Universal Robots URScript: proiecFinalHILT_cri.script

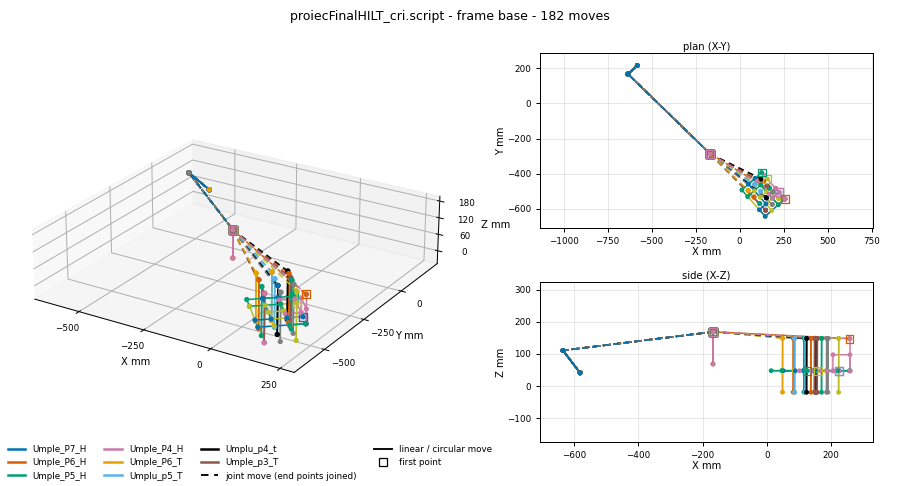
[picture p0: tool path of proiecFinalHILT_cri.script in frame base, 182 of 182 moves have a stored position in this frame; points joined in program order, loops and branches not executed]
def proiecFinalHILT_cri():
  set_gravity([0.0, 0.0, 9.82])
  set_safety_mode_transition_hardness(1)
  set_tool_voltage(24)
  set_tcp(p[0.0,0.0,0.27041000000000004,0.0,0.0,0.0])
  set_payload(0.9, [0.0, 0.0, 0.17])
  set_standard_analog_input_domain(0, 1)
  set_standard_analog_input_domain(1, 1)
  set_tool_analog_input_domain(0, 1)
  set_tool_analog_input_domain(1, 1)
  set_analog_outputdomain(0, 0)
  set_analog_outputdomain(1, 0)
  set_input_actions_to_default()
  step_count_8b5a3645_88be_4d1b_a3a9_0bb7bcbc2ce0 = 0.0
  thread Step_Counter_Thread_93ffaa2a_25e0_4f6a_ae18_d9d09f0d3b97():
    while (True):
      step_count_8b5a3645_88be_4d1b_a3a9_0bb7bcbc2ce0 = step_count_8b5a3645_88be_4d1b_a3a9_0bb7bcbc2ce0 + 1.0
      sync()
    end
  end
  run Step_Counter_Thread_93ffaa2a_25e0_4f6a_ae18_d9d09f0d3b97()
  global poz_switch=3
  global Dist_cub=80
  global countt=2
  global lp=5
  global i_var_1=6
  global Cub=p[-0.5333733899169065,0.2215163955594962,0.16621704113782268,0.29676891717628096,-0.762003058255801,0.6932450754498153]
  global Masa=p[-0.5646864889252723,-0.09295846005778519,-0.011586725889142446,-0.002204506099067434,-1.5199745422116683E-4,-0.8484235711542728]
  global Perete=p[0.07880424455785079,-0.9029855161661187,0.02758526437122058,1.5020481596863833,0.5702478707698211,0.5632393139112222]
  global plan_masa=p[-0.5631648595800378,-0.0915378818255476,-0.042707498643383746,-0.004205331887450723,8.438780583721072E-4,-0.8451230678381721]
  def Umple_P7_H():
    $ 52 "Umple_P7_H" "noBreak"
    $ 53 "MoveJ"
    $ 54 "INTERMED_P7_H" "breakAfter"
    movej(get_inverse_kin(p[-.167567487318, -.286498978533, .168810821008, 1.290941150555, 2.847903107563, -.014389347024], qnear=[0.6869624853134155, -1.9919636885272425, 1.8788256645202637, -1.4593976179706019, -1.5535171667682093, -0.03263694444765264]), a=1.3962634015954636, v=1.0471975511965976)
    $ 55 "Wait: 0.5"
    sleep(0.5)
    $ 56 "MoveJ"
    $ 57 "DEAS_C7_H" "breakAfter"
    movej(get_inverse_kin(p[-.634048678821, .166752753814, .111017315668, 1.076095386128, 2.388610774545, 1.006493672938], qnear=[-0.13465482393373662, -0.5505560080157679, 0.2975288927555084, -0.7133148352252405, -2.1372297445880335, -0.6779091993915003]), a=1.3962634015954636, v=1.0471975511965976)
    $ 58 "Wait: 0.5"
    sleep(0.5)
    $ 59 "MoveL"
    $ 60 "PREL_C7_H" "breakAfter"
    movel(p[-.580966948563, .215040941302, .041371233320, 1.076095361124, 2.388610928008, 1.006493864198], a=1.2, v=0.25)
    $ 61 "Wait: 0.5"
    sleep(0.5)
    $ 62 "'G40'"
    # 'G40'
    $ 63 "MoveL"
    $ 64 "DEAS_C7_HH" "breakAfter"
    movel(p[-.634048678821, .166752753814, .111017315668, 1.076095386128, 2.388610774545, 1.006493672938], a=1.2, v=0.25)
    $ 65 "Wait: 0.5"
    sleep(0.5)
    $ 66 "MoveJ"
    $ 67 "intermed" "breakAfter"
    movej(get_inverse_kin(p[-.167567487318, -.286498978533, .168810821008, 1.290941150555, 2.847903107563, -.014389347024], qnear=[0.6869624853134155, -1.9919636885272425, 1.8788256645202637, -1.4593976179706019, -1.5535171667682093, -0.03263694444765264]), a=1.3962634015954636, v=1.0471975511965976)
    $ 68 "Wait: 0.5"
    sleep(0.5)
    $ 69 "MoveJ"
    $ 70 "DEAS_P7_H_FOAIE" "breakAfter"
    movej(get_inverse_kin(p[.152399925349, -.536216503558, .148554934455, 1.291226875826, 2.847366244409, -.014273160143], qnear=[1.6449040174484253, -1.443597141896383, 1.4715391397476196, -1.6139887014972132, -1.5619214216815394, 0.9256654977798462]), a=1.3962634015954636, v=1.0471975511965976)
    $ 71 "Wait: 0.5"
    sleep(0.5)
    $ 72 "MoveJ"
    $ 73 "LAS_P7_H_FOAIE" "breakAfter"
    movej(get_inverse_kin(p[.151994766277, -.536783252620, -.018790607241, 1.291226898298, 2.847366305883, -.014273512506], qnear=[1.6440799236297607, -1.3487656752215784, 1.8007179498672485, -2.0379918257342737, -1.561909023915426, 0.9248414635658264]), a=1.3962634015954636, v=1.0471975511965976)
    $ 74 "Wait: 0.5"
    sleep(0.5)
    $ 75 "'G 80'"
    # 'G 80'
    $ 76 "MoveL"
    $ 77 "DEAS_C7_H_FOAIE" "breakAfter"
    movel(p[.152399925349, -.536216503558, .148554934455, 1.291226875826, 2.847366244409, -.014273160143], a=1.2, v=0.25)
  end
  def Umple_P6_H():
    $ 78 "Umple_P6_H" "noBreak"
    $ 79 "MoveJ"
    $ 80 "INTERM_C6_H" "breakAfter"
    movej(get_inverse_kin(p[-.167567487318, -.286498978533, .168810821008, 1.290941150555, 2.847903107563, -.014389347024], qnear=[0.6869624853134155, -1.9919636885272425, 1.8788256645202637, -1.4593976179706019, -1.5535171667682093, -0.03263694444765264]), a=1.3962634015954636, v=1.0471975511965976)
    $ 81 "Wait: 0.5"
    sleep(0.5)
    $ 82 "MoveJ"
    $ 83 "DEAS_C6_H" "breakAfter"
    movej(get_inverse_kin(p[-.634048678821, .166752753814, .111017315668, 1.076095386128, 2.388610774545, 1.006493672938], qnear=[-0.13465482393373662, -0.5505560080157679, 0.2975288927555084, -0.7133148352252405, -2.1372297445880335, -0.6779091993915003]), a=1.3962634015954636, v=1.0471975511965976)
    $ 84 "Wait: 0.5"
    sleep(0.5)
    $ 85 "MoveL"
    $ 86 "PREL_C6_H" "breakAfter"
    movel(p[-.580966948563, .215040941302, .041371233320, 1.076095361124, 2.388610928008, 1.006493864198], a=1.2, v=0.25)
    $ 87 "Wait: 0.5"
    sleep(0.5)
    $ 88 "'G40'"
    # 'G40'
    $ 89 "MoveL"
    $ 90 "DEAS_C6_HH" "breakAfter"
    movel(p[-.634048678821, .166752753814, .111017315668, 1.076095386128, 2.388610774545, 1.006493672938], a=1.2, v=0.25)
    $ 91 "Wait: 0.5"
    sleep(0.5)
    $ 92 "MoveJ"
    $ 93 "INTERMEDIARR" "breakAfter"
    movej(get_inverse_kin(p[-.167567487318, -.286498978533, .168810821008, 1.290941150555, 2.847903107563, -.014389347024], qnear=[0.6869624853134155, -1.9919636885272425, 1.8788256645202637, -1.4593976179706019, -1.5535171667682093, -0.03263694444765264]), a=1.3962634015954636, v=1.0471975511965976)
    $ 94 "Wait: 0.5"
    sleep(0.5)
    $ 95 "MoveJ"
    $ 96 "DEAS_P6_H_FOAIE" "breakAfter"
    movej(get_inverse_kin(p[.081815537007, -.531995464645, .148711679169, 2.983820748964, .973323486254, -.005655071201], qnear=[1.5207152366638184, -1.4787958304034632, 1.5076936483383179, -1.6038115660296839, -1.5730794111834925, 2.4608724117279053]), a=1.3962634015954636, v=1.0471975511965976)
    $ 97 "Wait: 0.5"
    sleep(0.5)
    $ 98 "MoveL"
    $ 99 "LAS_P6_H_FOAIE" "breakAfter"
    movel(p[.081410644423, -.532561926736, -.018634025734, 2.983821082689, .973324781842, -.005655577080], a=1.2, v=0.25)
    $ 100 "Wait: 0.5"
    sleep(0.5)
    $ 101 "'G 80'"
    # 'G 80'
    $ 102 "MoveL"
    $ 103 "DEAS_C6_H_FOAIE" "breakAfter"
    movel(p[.081815486859, -.531995349178, .148711350252, 2.983819433937, .973322093540, -.005646498257], a=1.2, v=0.25)
    $ 104 "Wait: 0.5"
    sleep(0.5)
  end
  def Umple_P5_H():
    $ 105 "Umple_P5_H" "noBreak"
    $ 106 "MoveJ"
    $ 107 "INTERM_P5_H" "breakAfter"
    movej(get_inverse_kin(p[-.167567487318, -.286498978533, .168810821008, 1.290941150555, 2.847903107563, -.014389347024], qnear=[0.6869624853134155, -1.9919636885272425, 1.8788256645202637, -1.4593976179706019, -1.5535171667682093, -0.03263694444765264]), a=1.3962634015954636, v=1.0471975511965976)
    $ 108 "Wait: 0.5"
    sleep(0.5)
    $ 109 "MoveJ"
    $ 110 "DEAS_C5_H" "breakAfter"
    movej(get_inverse_kin(p[-.634048678821, .166752753814, .111017315668, 1.076095386128, 2.388610774545, 1.006493672938], qnear=[-0.13465482393373662, -0.5505560080157679, 0.2975288927555084, -0.7133148352252405, -2.1372297445880335, -0.6779091993915003]), a=1.3962634015954636, v=1.0471975511965976)
    $ 111 "Wait: 0.5"
    sleep(0.5)
    $ 112 "MoveL"
    $ 113 "PREL_C5_H" "breakAfter"
    movel(p[-.580966948563, .215040941302, .041371233320, 1.076095361124, 2.388610928008, 1.006493864198], a=1.2, v=0.25)
    $ 114 "Wait: 0.5"
    sleep(0.5)
    $ 115 "'G40'"
    # 'G40'
    $ 116 "MoveL"
    $ 117 "DEAS_C5_HH" "breakAfter"
    movel(p[-.634048678821, .166752753814, .111017315668, 1.076095386128, 2.388610774545, 1.006493672938], a=1.2, v=0.25)
    $ 118 "Wait: 0.5"
    sleep(0.5)
    $ 119 "MoveJ"
    $ 120 "inter" "breakAfter"
    movej(get_inverse_kin(p[-.167567487318, -.286498978533, .168810821008, 1.290941150555, 2.847903107563, -.014389347024], qnear=[0.6869624853134155, -1.9919636885272425, 1.8788256645202637, -1.4593976179706019, -1.5535171667682093, -0.03263694444765264]), a=1.3962634015954636, v=1.0471975511965976)
    $ 121 "Wait: 0.5"
    sleep(0.5)
    $ 122 "MoveJ"
    $ 123 "DEAS_P5_H_FOAIE" "breakAfter"
    movej(get_inverse_kin(p[.114997524645, -.569397994153, .148757924677, 2.983821051292, .973323637050, -.005654878888], qnear=[1.582621455192566, -1.3755558172809046, 1.388292908668518, -1.587501351033346, -1.5733297506915491, 2.522778272628784]), a=1.3962634015954636, v=1.0471975511965976)
    $ 124 "Wait: 0.5"
    sleep(0.5)
    $ 125 "MoveL"
    $ 126 "LAS_P5_H_FOAIE" "breakAfter"
    movel(p[.114592639963, -.569964547732, -.018587646533, 2.983820983248, .973324799820, -.005655526622], a=1.2, v=0.25)
    $ 127 "Wait: 0.5"
    sleep(0.5)
    $ 128 "'G 80'"
    # 'G 80'
    $ 129 "MoveL"
    $ 130 "DEAS_C5_H_FOAIE" "breakAfter"
    movel(p[.114997433899, -.569398004731, .148757767474, 2.983819195458, .973322065302, -.005646601422], a=1.2, v=0.25)
    $ 131 "Wait: 0.5"
    sleep(0.5)
  end
  def Umple_P4_H():
    $ 132 "Umple_P4_H" "noBreak"
    $ 133 "MoveJ"
    $ 134 "INTERM_P4_H" "breakAfter"
    movej(get_inverse_kin(p[-.167567487318, -.286498978533, .168810821008, 1.290941150555, 2.847903107563, -.014389347024], qnear=[0.6869624853134155, -1.9919636885272425, 1.8788256645202637, -1.4593976179706019, -1.5535171667682093, -0.03263694444765264]), a=1.3962634015954636, v=1.0471975511965976)
    $ 135 "Wait: 0.5"
    sleep(0.5)
    $ 136 "MoveJ"
    $ 137 "DEAS_C4_H" "breakAfter"
    movej(get_inverse_kin(p[-.634048678821, .166752753814, .111017315668, 1.076095386128, 2.388610774545, 1.006493672938], qnear=[-0.13465482393373662, -0.5505560080157679, 0.2975288927555084, -0.7133148352252405, -2.1372297445880335, -0.6779091993915003]), a=1.3962634015954636, v=1.0471975511965976)
    $ 138 "Wait: 0.5"
    sleep(0.5)
    $ 139 "MoveL"
    $ 140 "PREL_C4_H" "breakAfter"
    movel(p[-.580966948563, .215040941302, .041371233320, 1.076095361124, 2.388610928008, 1.006493864198], a=1.2, v=0.25)
    $ 141 "Wait: 0.5"
    sleep(0.5)
    $ 142 "'G40'"
    # 'G40'
    $ 143 "MoveL"
    $ 144 "DEAS_C4_HH" "breakAfter"
    movel(p[-.634048678821, .166752753814, .111017315668, 1.076095386128, 2.388610774545, 1.006493672938], a=1.2, v=0.25)
    $ 145 "Wait: 0.5"
    sleep(0.5)
    $ 146 "MoveJ"
    $ 147 "INTERMEDIA" "breakAfter"
    movej(get_inverse_kin(p[-.167567487318, -.286498978533, .168810821008, 1.290941150555, 2.847903107563, -.014389347024], qnear=[0.6869624853134155, -1.9919636885272425, 1.8788256645202637, -1.4593976179706019, -1.5535171667682093, -0.03263694444765264]), a=1.3962634015954636, v=1.0471975511965976)
    $ 148 "Wait: 0.5"
    sleep(0.5)
    $ 149 "MoveJ"
    $ 150 "DEAS_P4_H_FOAIE" "breakAfter"
    movej(get_inverse_kin(p[.148179526257, -.606800607225, .148804148337, 2.983821216675, .973323524331, -.005654610012], qnear=[1.6362345218658447, -1.2673490683185022, 1.2510157823562622, -1.5582893530475062, -1.573538605366842, 2.5763912200927734]), a=1.3962634015954636, v=1.0471975511965976)
    $ 151 "Wait: 0.5"
    sleep(0.5)
    $ 152 "MoveL"
    $ 153 "LAS_P4_H_FOAIE" "breakAfter"
    movel(p[.147774535974, -.607367175758, -.018541400911, 2.983821119944, .973324675130, -.005655864895], a=1.2, v=0.25)
    $ 154 "Wait: 0.5"
    sleep(0.5)
    $ 155 "'G 80'"
    # 'G 80'
    $ 156 "MoveL"
    $ 157 "DEAS_P4_H" "breakAfter"
    movel(p[.148179486526, -.606800539344, .148804102555, 2.983819245133, .973322110034, -.005646290070], a=1.2, v=0.25)
    $ 158 "Wait: 0.5"
    sleep(0.5)
  end
  def Umple_P6_T():
    $ 159 "Umple_P6_T" "noBreak"
    $ 160 "MoveJ"
    $ 161 "INTERM_C6_T" "breakAfter"
    movej(get_inverse_kin(p[-.167567487318, -.286498978533, .168810821008, 1.290941150555, 2.847903107563, -.014389347024], qnear=[0.6869624853134155, -1.9919636885272425, 1.8788256645202637, -1.4593976179706019, -1.5535171667682093, -0.03263694444765264]), a=1.3962634015954636, v=1.0471975511965976)
    $ 162 "Wait: 0.5"
    sleep(0.5)
    $ 163 "MoveJ"
    $ 164 "DEAS_C6_T" "breakAfter"
    movej(get_inverse_kin(p[-.634048678821, .166752753814, .111017315668, 1.076095386128, 2.388610774545, 1.006493672938], qnear=[-0.13465482393373662, -0.5505560080157679, 0.2975288927555084, -0.7133148352252405, -2.1372297445880335, -0.6779091993915003]), a=1.3962634015954636, v=1.0471975511965976)
    $ 165 "Wait: 0.5"
    sleep(0.5)
    $ 166 "MoveL"
    $ 167 "PREL_C6_T" "breakAfter"
    movel(p[-.580966948563, .215040941302, .041371233320, 1.076095361124, 2.388610928008, 1.006493864198], a=1.2, v=0.25)
    $ 168 "Wait: 0.5"
    sleep(0.5)
    $ 169 "'G40'"
    # 'G40'
    $ 170 "MoveL"
    $ 171 "DEAS_C6_TT" "breakAfter"
    movel(p[-.634048678821, .166752753814, .111017315668, 1.076095386128, 2.388610774545, 1.006493672938], a=1.2, v=0.25)
    $ 172 "Wait: 0.5"
    sleep(0.5)
    $ 173 "MoveJ"
    $ 174 "INTERME" "breakAfter"
    movej(get_inverse_kin(p[-.167567487318, -.286498978533, .168810821008, 1.290941150555, 2.847903107563, -.014389347024], qnear=[0.6869624853134155, -1.9919636885272425, 1.8788256645202637, -1.4593976179706019, -1.5535171667682093, -0.03263694444765264]), a=1.3962634015954636, v=1.0471975511965976)
    $ 175 "Wait: 0.5"
    sleep(0.5)
    $ 176 "MoveJ"
    $ 177 "DEAS_P6_T_FOAIE" "breakAfter"
    movej(get_inverse_kin(p[.086036154554, -.461411134347, .148462036457, 2.983821038078, .973324356096, -.005654006834], qnear=[1.5222129821777344, -1.644914452229635, 1.676056146621704, -1.606051270161764, -1.573085133229391, 2.462369680404663]), a=1.3962634015954636, v=1.0471975511965976)
    $ 178 "Wait: 0.5"
    sleep(0.5)
    $ 179 "MoveL"
    $ 180 "LAS_C6_T_FOAIE" "breakAfter"
    movel(p[.085630996758, -.461978027654, -.018883318685, 2.983820678969, .973324049014, -.005654378319], a=1.2, v=0.25)
    $ 181 "Wait: 0.5"
    sleep(0.5)
    $ 182 "'G 80'"
    # 'G 80'
    $ 183 "MoveL"
    $ 184 "DEAS_P6_T" "breakAfter"
    movel(p[.086036154554, -.461411134347, .148462036457, 2.983821038078, .973324356096, -.005654006834], a=1.2, v=0.25)
    $ 185 "Wait: 0.5"
    sleep(0.5)
  end
  def Umplu_p5_T():
    $ 186 "Umplu_p5_T" "noBreak"
    $ 187 "MoveJ"
    $ 188 "INTERM_P5_T" "breakAfter"
    movej(get_inverse_kin(p[-.167567487318, -.286498978533, .168810821008, 1.290941150555, 2.847903107563, -.014389347024], qnear=[0.6869624853134155, -1.9919636885272425, 1.8788256645202637, -1.4593976179706019, -1.5535171667682093, -0.03263694444765264]), a=1.3962634015954636, v=1.0471975511965976)
    $ 189 "Wait: 0.5"
    sleep(0.5)
    $ 190 "MoveJ"
    $ 191 "DEAS_C5_T" "breakAfter"
    movej(get_inverse_kin(p[-.634048678821, .166752753814, .111017315668, 1.076095386128, 2.388610774545, 1.006493672938], qnear=[-0.13465482393373662, -0.5505560080157679, 0.2975288927555084, -0.7133148352252405, -2.1372297445880335, -0.6779091993915003]), a=1.3962634015954636, v=1.0471975511965976)
    $ 192 "Wait: 0.5"
    sleep(0.5)
    $ 193 "MoveL"
    $ 194 "PREL_C5_T" "breakAfter"
    movel(p[-.580966948563, .215040941302, .041371233320, 1.076095361124, 2.388610928008, 1.006493864198], a=1.2, v=0.25)
    $ 195 "Wait: 0.5"
    sleep(0.5)
    $ 196 "'G40'"
    # 'G40'
    $ 197 "MoveL"
    $ 198 "DEAS_C5_TT" "breakAfter"
    movel(p[-.634048678821, .166752753814, .111017315668, 1.076095386128, 2.388610774545, 1.006493672938], a=1.2, v=0.25)
    $ 199 "Wait: 0.5"
    sleep(0.5)
    $ 200 "MoveJ"
    $ 201 "INter" "breakAfter"
    movej(get_inverse_kin(p[-.167567487318, -.286498978533, .168810821008, 1.290941150555, 2.847903107563, -.014389347024], qnear=[0.6869624853134155, -1.9919636885272425, 1.8788256645202637, -1.4593976179706019, -1.5535171667682093, -0.03263694444765264]), a=1.3962634015954636, v=1.0471975511965976)
    $ 202 "Wait: 0.5"
    sleep(0.5)
    $ 203 "MoveJ"
    $ 204 "DEAS_P5_T_FOAIE" "breakAfter"
    movej(get_inverse_kin(p[.119218109273, -.498813767404, .148508400157, 2.983820953563, .973324318096, -.005654075141], qnear=[1.592743992805481, -1.5396392981158655, 1.5730714797973633, -1.6081703344928187, -1.57336932817568, 2.532900333404541]), a=1.3962634015954636, v=1.0471975511965976)
    $ 205 "Wait: 0.5"
    sleep(0.5)
    $ 206 "MoveL"
    $ 207 "LAS_C5_T_FOAIE" "breakAfter"
    movel(p[.118812995133, -.499380619453, -.018837005131, 2.983820836474, .973323892156, -.005654109965], a=1.2, v=0.25)
    $ 208 "Wait: 0.5"
    sleep(0.5)
    $ 209 "'G 80'"
    # 'G 80'
    $ 210 "MoveL"
    $ 211 "DEAS_P5" "breakAfter"
    movel(p[.119218109273, -.498813767404, .148508400157, 2.983820953563, .973324318096, -.005654075141], a=1.2, v=0.25)
    $ 212 "Wait: 0.5"
    sleep(0.5)
  end
  def Umplu_p4_t():
    $ 213 "Umplu_p4_t" "noBreak"
    $ 214 "MoveJ"
    $ 215 "interm_p4_t" "breakAfter"
    movej(get_inverse_kin(p[-.167567487318, -.286498978533, .168810821008, 1.290941150555, 2.847903107563, -.014389347024], qnear=[0.6869624853134155, -1.9919636885272425, 1.8788256645202637, -1.4593976179706019, -1.5535171667682093, -0.03263694444765264]), a=1.3962634015954636, v=1.0471975511965976)
    $ 216 "Wait: 0.5"
    sleep(0.5)
    $ 217 "MoveJ"
    $ 218 "deas_c4_T" "breakAfter"
    movej(get_inverse_kin(p[-.634048678821, .166752753814, .111017315668, 1.076095386128, 2.388610774545, 1.006493672938], qnear=[-0.13465482393373662, -0.5505560080157679, 0.2975288927555084, -0.7133148352252405, -2.1372297445880335, -0.6779091993915003]), a=1.3962634015954636, v=1.0471975511965976)
    $ 219 "Wait: 0.5"
    sleep(0.5)
    $ 220 "MoveL"
    $ 221 "PREL_C4_T" "breakAfter"
    movel(p[-.580966948563, .215040941302, .041371233320, 1.076095361124, 2.388610928008, 1.006493864198], a=1.2, v=0.25)
    $ 222 "Wait: 0.5"
    sleep(0.5)
    $ 223 "'G40'"
    # 'G40'
    $ 224 "MoveL"
    $ 225 "DEAS_C4_T" "breakAfter"
    movel(p[-.634048678821, .166752753814, .111017315668, 1.076095386128, 2.388610774545, 1.006493672938], a=1.2, v=0.25)
    $ 226 "Wait: 0.5"
    sleep(0.5)
    $ 227 "MoveJ"
    $ 228 "INTERMEDIAR" "breakAfter"
    movej(get_inverse_kin(p[-.167567487318, -.286498978533, .168810821008, 1.290941150555, 2.847903107563, -.014389347024], qnear=[0.6869624853134155, -1.9919636885272425, 1.8788256645202637, -1.4593976179706019, -1.5535171667682093, -0.03263694444765264]), a=1.3962634015954636, v=1.0471975511965976)
    $ 229 "Wait: 0.5"
    sleep(0.5)
    $ 230 "MoveJ"
    $ 231 "DEAS_P4_T_FOAIE" "breakAfter"
    movej(get_inverse_kin(p[.152399990844, -.536216423213, .148554701618, 2.983821087416, .973324179283, -.005654354735], qnear=[1.652442216873169, -1.4321559111224573, 1.4555567502975464, -1.597978417073385, -1.5736001173602503, 2.5925984382629395]), a=1.3962634015954636, v=1.0471975511965976)
    $ 232 "Wait: 0.5"
    sleep(0.5)
    $ 233 "MoveL"
    $ 234 "LAS_P4_T_FOAIE" "breakAfter"
    movel(p[.151994974835, -.536783166276, -.018790624961, 2.983820916063, .973323931244, -.005654087772], a=1.2, v=0.25)
    $ 235 "Wait: 0.5"
    sleep(0.5)
    $ 236 "'G 80'"
    # 'G 80'
    $ 237 "MoveL"
    $ 238 "DEAS_P4_T" "breakAfter"
    movel(p[.152399990844, -.536216423213, .148554701618, 2.983821087416, .973324179283, -.005654354735], a=1.2, v=0.25)
    $ 239 "Wait: 0.5"
    sleep(0.5)
  end
  def Umple_p3_T():
    $ 240 "Umple_p3_T" "noBreak"
    $ 241 "MoveJ"
    $ 242 "INTERM_P3_T" "breakAfter"
    movej(get_inverse_kin(p[-.167567487318, -.286498978533, .168810821008, 1.290941150555, 2.847903107563, -.014389347024], qnear=[0.6869624853134155, -1.9919636885272425, 1.8788256645202637, -1.4593976179706019, -1.5535171667682093, -0.03263694444765264]), a=1.3962634015954636, v=1.0471975511965976)
    $ 243 "Wait: 0.5"
    sleep(0.5)
    $ 244 "MoveJ"
    $ 245 "DEAS_C3_T" "breakAfter"
    movej(get_inverse_kin(p[-.634048678821, .166752753814, .111017315668, 1.076095386128, 2.388610774545, 1.006493672938], qnear=[-0.13465482393373662, -0.5505560080157679, 0.2975288927555084, -0.7133148352252405, -2.1372297445880335, -0.6779091993915003]), a=1.3962634015954636, v=1.0471975511965976)
    $ 246 "Wait: 0.5"
    sleep(0.5)
    $ 247 "MoveL"
    $ 248 "PREL_C3_T" "breakAfter"
    movel(p[-.580966948563, .215040941302, .041371233320, 1.076095361124, 2.388610928008, 1.006493864198], a=1.2, v=0.25)
    $ 249 "Wait: 0.5"
    sleep(0.5)
    $ 250 "'G40'"
    # 'G40'
    $ 251 "MoveL"
    $ 252 "DEAS_C3_TT" "breakAfter"
    movel(p[-.634048678821, .166752753814, .111017315668, 1.076095386128, 2.388610774545, 1.006493672938], a=1.2, v=0.25)
    $ 253 "Wait: 0.5"
    sleep(0.5)
    $ 254 "MoveJ"
    $ 255 "INTERMEDD" "breakAfter"
    movej(get_inverse_kin(p[-.167567487318, -.286498978533, .168810821008, 1.290941150555, 2.847903107563, -.014389347024], qnear=[0.6869624853134155, -1.9919636885272425, 1.8788256645202637, -1.4593976179706019, -1.5535171667682093, -0.03263694444765264]), a=1.3962634015954636, v=1.0471975511965976)
    $ 256 "Wait: 0.5"
    sleep(0.5)
    $ 257 "MoveJ"
    $ 258 "DEAS_P3_T_FOAIE" "breakAfter"
    movej(get_inverse_kin(p[.148179528223, -.606800592740, .148804018507, 1.291225298432, 2.847366483862, -.014273607498], qnear=[1.6294351816177368, -1.2790477911578577, 1.2692852020263672, -1.5761454741107386, -1.5616863409625452, 0.910196840763092]), a=1.3962634015954636, v=1.0471975511965976)
    $ 259 "Wait: 0.5"
    sleep(0.5)
    $ 260 "MoveL"
    $ 261 "LAS_P3_T_FOAIE" "breakAfter"
    movel(p[.147774525895, -.607367213899, -.018541509057, 1.291225168160, 2.847366616510, -.014273004499], a=1.2, v=0.25)
    $ 262 "Wait: 0.5"
    sleep(0.5)
    $ 263 "'G 80'"
    # 'G 80'
    $ 264 "MoveL"
    $ 265 "DEAS_P3_T" "breakAfter"
    movel(p[.148179528223, -.606800592740, .148804018507, 1.291225298432, 2.847366483862, -.014273607498], a=1.2, v=0.25)
    $ 266 "Wait: 0.5"
    sleep(0.5)
  end
  def Umple_P2_T():
    $ 267 "Umple_P2_T" "noBreak"
    $ 268 "MoveJ"
    $ 269 "INTERM_P2_T" "breakAfter"
    movej(get_inverse_kin(p[-.167567487318, -.286498978533, .168810821008, 1.290941150555, 2.847903107563, -.014389347024], qnear=[0.6869624853134155, -1.9919636885272425, 1.8788256645202637, -1.4593976179706019, -1.5535171667682093, -0.03263694444765264]), a=1.3962634015954636, v=1.0471975511965976)
    $ 270 "Wait: 0.5"
    sleep(0.5)
    $ 271 "MoveJ"
    $ 272 "DEAS_P2_T" "breakAfter"
    movej(get_inverse_kin(p[-.634048678821, .166752753814, .111017315668, 1.076095386128, 2.388610774545, 1.006493672938], qnear=[-0.13465482393373662, -0.5505560080157679, 0.2975288927555084, -0.7133148352252405, -2.1372297445880335, -0.6779091993915003]), a=1.3962634015954636, v=1.0471975511965976)
    $ 273 "Wait: 0.5"
    sleep(0.5)
    $ 274 "MoveL"
    $ 275 "PREL_C2_T" "breakAfter"
    movel(p[-.580966948563, .215040941302, .041371233320, 1.076095361124, 2.388610928008, 1.006493864198], a=1.2, v=0.25)
    $ 276 "Wait: 0.5"
    sleep(0.5)
    $ 277 "'G40'"
    # 'G40'
    $ 278 "MoveL"
    $ 279 "DEAS_C2_T" "breakAfter"
    movel(p[-.634048678821, .166752753814, .111017315668, 1.076095386128, 2.388610774545, 1.006493672938], a=1.2, v=0.25)
    $ 280 "Wait: 0.5"
    sleep(0.5)
    $ 281 "MoveJ"
    $ 282 "INTERMED" "breakAfter"
    movej(get_inverse_kin(p[-.167567487318, -.286498978533, .168810821008, 1.290941150555, 2.847903107563, -.014389347024], qnear=[0.6869624853134155, -1.9919636885272425, 1.8788256645202637, -1.4593976179706019, -1.5535171667682093, -0.03263694444765264]), a=1.3962634015954636, v=1.0471975511965976)
    $ 283 "Wait: 0.5"
    sleep(0.5)
    $ 284 "MoveJ"
    $ 285 "DEAS_P2_T_FOAIE" "breakAfter"
    movej(get_inverse_kin(p[.185581949577, -.573618939446, .148601050831, 1.291225391927, 2.847366587857, -.014273246615], qnear=[1.696845293045044, -1.3333137671100062, 1.339584231376648, -1.592757527028219, -1.5627248922931116, 0.9776014685630798]), a=1.3962634015954636, v=1.0471975511965976)
    $ 286 "Wait: 0.5"
    sleep(0.5)
    $ 287 "MoveL"
    $ 288 "LAS_P2_T_FOAIE" "breakAfter"
    movel(p[.185176974658, -.574185681297, -.018744368520, 1.291225186600, 2.847366418911, -.014273142291], a=1.2, v=0.25)
    $ 289 "Wait: 0.5"
    sleep(0.5)
    $ 290 "'G 80'"
    # 'G 80'
    $ 291 "MoveL"
    $ 292 "DEAS_P2_T_F" "breakAfter"
    movel(p[.185581949577, -.573618939446, .148601050831, 1.291225391927, 2.847366587857, -.014273246615], a=1.2, v=0.25)
    $ 293 "Wait: 0.5"
    sleep(0.5)
  end
  def Desen_H():
    $ 294 "Desen_H" "noBreak"
    $ 295 "MoveL"
    $ 296 "L1_H" "breakAfter"
    movel(p[.158353767573, -.430155299332, .047611332993, 1.296043145667, 2.848527183735, .014471728358], a=1.2, v=0.25)
    $ 297 "MoveL"
    $ 298 "L2_H" "breakAfter"
    movel(p[.120951283833, -.463336924786, .047814223162, 1.296043120148, 2.848527345096, .014471416584], a=1.2, v=0.25)
    $ 299 "MoveL"
    $ 300 "L3_H" "breakAfter"
    movel(p[.154133236674, -.500739444601, .047860495744, 1.296043187324, 2.848527522418, .014471774946], a=1.2, v=0.25)
    $ 301 "MoveL"
    $ 302 "L4_H" "breakAfter"
    movel(p[.116730864622, -.533921061136, .048063444108, 1.296043121592, 2.848527328027, .014471677397], a=1.2, v=0.25)
    $ 303 "MoveL"
    $ 304 "L5_H" "breakAfter"
    movel(p[.083548907102, -.496518450929, .048017030358, 1.296043098946, 2.848527421426, .014471904572], a=1.2, v=0.25)
    $ 305 "MoveL"
    $ 306 "L6_H" "breakAfter"
    movel(p[.046146485395, -.529699970965, .048219970789, 1.296043094495, 2.848527467819, .014471901899], a=1.2, v=0.25)
    $ 307 "MoveL"
    $ 308 "L7_H" "breakAfter"
    movel(p[.145692315173, -.641907763135, .048359070968, 1.296043194804, 2.848527583583, .014471694291], a=1.2, v=0.25)
    $ 309 "MoveL"
    $ 310 "L8" "breakAfter"
    movel(p[.183094788894, -.608726180961, .048156303017, 1.296043066858, 2.848527509527, .014471421053], a=1.2, v=0.25)
    $ 311 "MoveL"
    $ 312 "L9_H" "breakAfter"
    movel(p[.149912797167, -.571323507272, .048109955944, 1.296043112977, 2.848527628353, .014471593212], a=1.2, v=0.25)
    $ 313 "MoveL"
    $ 314 "L10_H" "breakAfter"
    movel(p[.187315154740, -.538141973257, .047906982215, 1.296043228903, 2.848527813831, .014471559318], a=1.2, v=0.25)
    $ 315 "MoveL"
    $ 316 "L11_H" "breakAfter"
    movel(p[.220497113487, -.575544528094, .047953430580, 1.296043230770, 2.848527753786, .014471533520], a=1.2, v=0.25)
    $ 317 "MoveL"
    $ 318 "L12_H" "breakAfter"
    movel(p[.257899491601, -.542362921046, .047750448037, 1.296043415155, 2.848527963236, .014471718970], a=1.2, v=0.25)
  end
  def Desen_T():
    $ 319 "Desen_T" "noBreak"
    $ 320 "MoveL"
    $ 321 "l1_T" "breakAfter"
    movel(p[.224717745310, -.504960528950, .047704168521, 1.296043065165, 2.848526931384, .014471352058], a=1.2, v=0.25)
    $ 322 "MoveL"
    $ 323 "l2_T" "breakAfter"
    movel(p[.187315272317, -.538142086044, .047906973360, 1.296043149277, 2.848527197326, .014471477363], a=1.2, v=0.25)
    $ 324 "MoveL"
    $ 325 "l3_T" "breakAfter"
    movel(p[.087769321683, -.425934317539, .047767997329, 1.296043100195, 2.848527282499, .014471150240], a=1.2, v=0.25)
    $ 326 "MoveL"
    $ 327 "l4_T" "breakAfter"
    movel(p[.050366823128, -.459115956447, .047970927808, 1.296043197593, 2.848527294810, .014470760370], a=1.2, v=0.25)
    $ 328 "MoveL"
    $ 329 "l5_T" "breakAfter"
    movel(p[.149912749792, -.571323861062, .048110045365, 1.296043089492, 2.848527153310, .014470272402], a=1.2, v=0.25)
    $ 330 "MoveL"
    $ 331 "l6_T" "breakAfter"
    movel(p[.112510303828, -.604505478994, .048312930113, 1.296043108336, 2.848527098013, .014470239028], a=1.2, v=0.25)
    $ 332 "MoveL"
    $ 333 "l7_T" "breakAfter"
    movel(p[.145692254958, -.641908116683, .048359160323, 1.296043175969, 2.848527118698, .014470364418], a=1.2, v=0.25)
    $ 334 "MoveL"
    $ 335 "l8_T" "breakAfter"
    movel(p[.257899539344, -.542363388286, .047750527044, 1.296043062532, 2.848527225834, .014470116205], a=1.2, v=0.25)
  end
  def Umplu_p3_i():
    $ 336 "Umplu_p3_i" "noBreak"
    $ 337 "MoveJ"
    $ 338 "interm_p3" "breakAfter"
    movej(get_inverse_kin(p[-.167567487318, -.286498978533, .168810821008, 1.290941150555, 2.847903107563, -.014389347024], qnear=[0.6869624853134155, -1.9919636885272425, 1.8788256645202637, -1.4593976179706019, -1.5535171667682093, -0.03263694444765264]), a=1.3962634015954636, v=1.0471975511965976)
    $ 339 "Wait: 0.5"
    sleep(0.5)
    $ 340 "MoveJ"
    $ 341 "deas_c3_i" "breakAfter"
    movej(get_inverse_kin(p[-.634048678821, .166752753814, .111017315668, 1.076095386128, 2.388610774545, 1.006493672938], qnear=[-0.13465482393373662, -0.5505560080157679, 0.2975288927555084, -0.7133148352252405, -2.1372297445880335, -0.6779091993915003]), a=1.3962634015954636, v=1.0471975511965976)
    $ 342 "Wait: 0.5"
    sleep(0.5)
    $ 343 "MoveL"
    $ 344 "prel_3_i" "breakAfter"
    movel(p[-.580966948563, .215040941302, .041371233320, 1.076095361124, 2.388610928008, 1.006493864198], a=1.2, v=0.25)
    $ 345 "Wait: 0.5"
    sleep(0.5)
    $ 346 "'G40'"
    # 'G40'
    $ 347 "MoveL"
    $ 348 "deas_c3_ii" "breakAfter"
    movel(p[-.634048678821, .166752753814, .111017315668, 1.076095386128, 2.388610774545, 1.006493672938], a=1.2, v=0.25)
    $ 349 "Wait: 0.5"
    sleep(0.5)
    $ 350 "MoveJ"
    $ 351 "interm" "breakAfter"
    movej(get_inverse_kin(p[-.167567487318, -.286498978533, .168810821008, 1.290941150555, 2.847903107563, -.014389347024], qnear=[0.6869624853134155, -1.9919636885272425, 1.8788256645202637, -1.4593976179706019, -1.5535171667682093, -0.03263694444765264]), a=1.3962634015954636, v=1.0471975511965976)
    $ 352 "Wait: 0.5"
    sleep(0.5)
    $ 353 "MoveJ"
    $ 354 "deas_p3_i_foaie" "breakAfter"
    movej(get_inverse_kin(p[.136710917520, -.443190700033, .148277597898, 2.983706779009, .973287613512, -.005232679259], qnear=[1.6343494653701782, -1.6582220236407679, 1.688613772392273, -1.6050694624530237, -1.5732410589801233, 2.5745058059692383]), a=1.3962634015954636, v=1.0471975511965976)
    $ 355 "Wait: 0.5"
    sleep(0.5)
    $ 356 "MoveL"
    $ 357 "las_p3_i_foaie" "breakAfter"
    movel(p[.136306192414, -.443757445123, -.019067699712, 2.983706719795, .973287408143, -.005231154998], a=1.2, v=0.25)
    $ 358 "Wait: 0.5"
    sleep(0.5)
    $ 359 "'G 80'"
    # 'G 80'
    $ 360 "MoveL"
    $ 361 "deas_p3_i" "breakAfter"
    movel(p[.136710967595, -.443190640401, .148277539713, 2.983707061866, .973287115721, -.005232631375], a=1.2, v=0.25)
  end
  def Umplu_p2_i():
    $ 362 "Umplu_p2_i" "noBreak"
    $ 363 "MoveJ"
    $ 364 "interm_p2_i" "breakAfter"
    movej(get_inverse_kin(p[-.167567487318, -.286498978533, .168810821008, 1.290941150555, 2.847903107563, -.014389347024], qnear=[0.6869624853134155, -1.9919636885272425, 1.8788256645202637, -1.4593976179706019, -1.5535171667682093, -0.03263694444765264]), a=1.3962634015954636, v=1.0471975511965976)
    $ 365 "Wait: 0.5"
    sleep(0.5)
    $ 366 "MoveJ"
    $ 367 "deas_c2_i" "breakAfter"
    movej(get_inverse_kin(p[-.634048678821, .166752753814, .111017315668, 1.076095386128, 2.388610774545, 1.006493672938], qnear=[-0.13465482393373662, -0.5505560080157679, 0.2975288927555084, -0.7133148352252405, -2.1372297445880335, -0.6779091993915003]), a=1.3962634015954636, v=1.0471975511965976)
    $ 368 "Wait: 0.5"
    sleep(0.5)
    $ 369 "MoveL"
    $ 370 "prel_c2_i" "breakAfter"
    movel(p[-.580966948563, .215040941302, .041371233320, 1.076095361124, 2.388610928008, 1.006493864198], a=1.2, v=0.25)
    $ 371 "Wait: 0.5"
    sleep(0.5)
    $ 372 "'G40'"
    # 'G40'
    $ 373 "MoveL"
    $ 374 "deas_c2_i2" "breakAfter"
    movel(p[-.634048678821, .166752753814, .111017315668, 1.076095386128, 2.388610774545, 1.006493672938], a=1.2, v=0.25)
    $ 375 "Wait: 0.5"
    sleep(0.5)
    $ 376 "MoveJ"
    $ 377 "intermmm" "breakAfter"
    movej(get_inverse_kin(p[-.167567487318, -.286498978533, .168810821008, 1.290941150555, 2.847903107563, -.014389347024], qnear=[0.6869624853134155, -1.9919636885272425, 1.8788256645202637, -1.4593976179706019, -1.5535171667682093, -0.03263694444765264]), a=1.3962634015954636, v=1.0471975511965976)
    $ 378 "Wait: 0.5"
    sleep(0.5)
    $ 379 "MoveJ"
    $ 380 "Deas_P2_I_FOaie" "breakAfter"
    movej(get_inverse_kin(p[.169892934208, -.480593350924, .148323950518, 2.983706611248, .973287743483, -.005232594662], qnear=[1.696690559387207, -1.54694110551943, 1.5810078382492065, -1.6085847059832972, -1.5734780470477503, 2.6368465423583984]), a=1.3962634015954636, v=1.0471975511965976)
    $ 381 "Wait: 0.5"
    sleep(0.5)
    $ 382 "MoveL"
    $ 383 "las_P2_i_foaie" "breakAfter"
    movel(p[.169488097210, -.481159998853, -.019021462959, 2.983706968312, .973287474864, -.005231319054], a=1.2, v=0.25)
    $ 384 "Wait: 0.5"
    sleep(0.5)
    $ 385 "'G 80'"
    # 'G 80'
    $ 386 "MoveL"
    $ 387 "deas_p2_i" "breakAfter"
    movel(p[.169892986025, -.480593287420, .148323892346, 2.983706895626, .973287246212, -.005232558159], a=1.2, v=0.25)
  end
  def Desen_i():
    $ 388 "Desen_i" "noBreak"
    $ 389 "MoveL"
    $ 390 "Caciulita_i1" "breakAfter"
    movel(p[.224717722166, -.504960484151, .047704103504, 1.291226847034, 2.847366347327, -.014272085334], a=1.2, v=0.25)
    $ 391 "MoveL"
    $ 392 "Caciulita_i2" "breakAfter"
    movel(p[.187315226594, -.538142043484, .047906977082, 1.291227032284, 2.847366301756, -.014272118413], a=1.2, v=0.25)
    $ 393 "MoveL"
    $ 394 "caciulita_i3" "breakAfter"
    movel(p[.220497136640, -.575544671583, .047953560433, 1.291225944203, 2.847366585140, -.014274123381], a=1.2, v=0.25)
    $ 395 "MoveL"
    $ 396 "Caciulita_i4" "breakAfter"
    movel(p[.257899562405, -.542362928148, .047750267064, 1.291226593864, 2.847366752439, -.014272422908], a=1.2, v=0.25)
    $ 397 "MoveL"
    $ 398 "spatiere1_i" "breakAfter"
    movel(p[.258020743673, -.542193728640, .097750042331, 1.291224449561, 2.847366863892, -.014275606648], a=1.2, v=0.25)
    $ 399 "MoveL"
    $ 400 "spatiere2_i" "breakAfter"
    movel(p[.204929683954, -.482349502149, .097676031332, 1.291226728538, 2.847366079793, -.014272245406], a=1.2, v=0.25)
    $ 401 "MoveL"
    $ 402 "spatiere3_i" "breakAfter"
    movel(p[.204808597099, -.482518777578, .047676475167, 1.291226441140, 2.847366455616, -.014273107727], a=1.2, v=0.25)
    $ 403 "MoveL"
    $ 404 "coada_i1" "breakAfter"
    movel(p[.138444723852, -.407713504749, .047583847563, 1.291226332997, 2.847366307920, -.014273010711], a=1.2, v=0.25)
    $ 405 "MoveL"
    $ 406 "coada_i2" "breakAfter"
    movel(p[.101042232951, -.440895027094, .047786740412, 1.291226372130, 2.847366540430, -.014272971580], a=1.2, v=0.25)
    $ 407 "MoveL"
    $ 408 "coada_i3" "breakAfter"
    movel(p[.167406116273, -.515700163940, .047879477850, 1.291226451164, 2.847366681792, -.014273039441], a=1.2, v=0.25)
    $ 409 "MoveL"
    $ 410 "coada_i4" "breakAfter"
    movel(p[.204808616914, -.482518553621, .047676614829, 1.291226300396, 2.847366594866, -.014272954152], a=1.2, v=0.25)
  end
  def Umplu_P6_L():
    $ 411 "Umplu_P6_L" "noBreak"
    $ 412 "MoveJ"
    $ 413 "INTERM_P6" "breakAfter"
    movej(get_inverse_kin(p[-.167567487318, -.286498978533, .168810821008, 1.290941150555, 2.847903107563, -.014389347024], qnear=[0.6869624853134155, -1.9919636885272425, 1.8788256645202637, -1.4593976179706019, -1.5535171667682093, -0.03263694444765264]), a=1.3962634015954636, v=1.0471975511965976)
    $ 414 "Wait: 0.5"
    sleep(0.5)
    $ 415 "MoveJ"
    $ 416 "DEAS_C6_L" "breakAfter"
    movej(get_inverse_kin(p[-.634048678821, .166752753814, .111017315668, 1.076095386128, 2.388610774545, 1.006493672938], qnear=[-0.13465482393373662, -0.5505560080157679, 0.2975288927555084, -0.7133148352252405, -2.1372297445880335, -0.6779091993915003]), a=1.3962634015954636, v=1.0471975511965976)
    $ 417 "Wait: 0.5"
    sleep(0.5)
    $ 418 "MoveL"
    $ 419 "PREL_C6_L" "breakAfter"
    movel(p[-.580966948563, .215040941302, .041371233320, 1.076095361124, 2.388610928008, 1.006493864198], a=1.2, v=0.25)
    $ 420 "Wait: 0.5"
    sleep(0.5)
    $ 421 "'G40'"
    # 'G40'
    $ 422 "MoveL"
    $ 423 "DEAS_C6_LL" "breakAfter"
    movel(p[-.634048678821, .166752753814, .111017315668, 1.076095386128, 2.388610774545, 1.006493672938], a=1.2, v=0.25)
    $ 424 "Wait: 0.5"
    sleep(0.5)
    $ 425 "MoveJ"
    $ 426 "INTERRR" "breakAfter"
    movej(get_inverse_kin(p[-.167567487318, -.286498978533, .168810821008, 1.290941150555, 2.847903107563, -.014389347024], qnear=[0.6869624853134155, -1.9919636885272425, 1.8788256645202637, -1.4593976179706019, -1.5535171667682093, -0.03263694444765264]), a=1.3962634015954636, v=1.0471975511965976)
    $ 427 "Wait: 0.5"
    sleep(0.5)
    $ 428 "MoveJ"
    $ 429 "DEAS_P6_L_FOAIE" "breakAfter"
    movej(get_inverse_kin(p[.048633517896, -.494592854746, .148664829593, 1.291226778572, 2.847366116501, -.014272865868], qnear=[1.438780665397644, -1.5881570021258753, 1.623896837234497, -1.6196473280536097, -1.5589879194842737, 0.7195518612861633]), a=1.3962634015954636, v=1.0471975511965976)
    $ 430 "Wait: 0.5"
    sleep(0.5)
    $ 431 "MoveL"
    $ 432 "LAS_C6_L_FOAIE" "breakAfter"
    movel(p[.048228385021, -.495159383447, -.018680489355, 1.291225956508, 2.847366377697, -.014272733564], a=1.2, v=0.25)
    $ 433 "Wait: 0.5"
    sleep(0.5)
    $ 434 "'G 80'"
    # 'G 80'
    $ 435 "MoveL"
    $ 436 "DEAS_P6_L" "breakAfter"
    movel(p[.048633520797, -.494592795841, .148664781155, 1.291226852439, 2.847366245931, -.014269626748], a=1.2, v=0.25)
  end
  def Umplu_P5_L():
    $ 437 "Umplu_P5_L" "noBreak"
    $ 438 "MoveJ"
    $ 439 "INTERM_P5" "breakAfter"
    movej(get_inverse_kin(p[-.167567487318, -.286498978533, .168810821008, 1.290941150555, 2.847903107563, -.014389347024], qnear=[0.6869624853134155, -1.9919636885272425, 1.8788256645202637, -1.4593976179706019, -1.5535171667682093, -0.03263694444765264]), a=1.3962634015954636, v=1.0471975511965976)
    $ 440 "Wait: 0.5"
    sleep(0.5)
    $ 441 "MoveJ"
    $ 442 "DEAS_C5_L" "breakAfter"
    movej(get_inverse_kin(p[-.634048678821, .166752753814, .111017315668, 1.076095386128, 2.388610774545, 1.006493672938], qnear=[-0.13465482393373662, -0.5505560080157679, 0.2975288927555084, -0.7133148352252405, -2.1372297445880335, -0.6779091993915003]), a=1.3962634015954636, v=1.0471975511965976)
    $ 443 "Wait: 0.5"
    sleep(0.5)
    $ 444 "MoveL"
    $ 445 "PREL_C5_L" "breakAfter"
    movel(p[-.580966948563, .215040941302, .041371233320, 1.076095361124, 2.388610928008, 1.006493864198], a=1.2, v=0.25)
    $ 446 "Wait: 0.5"
    sleep(0.5)
    $ 447 "'G40'"
    # 'G40'
    $ 448 "MoveL"
    $ 449 "DEAS_C5_LL" "breakAfter"
    movel(p[-.634048678821, .166752753814, .111017315668, 1.076095386128, 2.388610774545, 1.006493672938], a=1.2, v=0.25)
    $ 450 "Wait: 0.5"
    sleep(0.5)
    $ 451 "MoveJ"
    $ 452 "INTERR" "breakAfter"
    movej(get_inverse_kin(p[-.167567487318, -.286498978533, .168810821008, 1.290941150555, 2.847903107563, -.014389347024], qnear=[0.6869624853134155, -1.9919636885272425, 1.8788256645202637, -1.4593976179706019, -1.5535171667682093, -0.03263694444765264]), a=1.3962634015954636, v=1.0471975511965976)
    $ 453 "Wait: 0.5"
    sleep(0.5)
    $ 454 "MoveJ"
    $ 455 "DEAS_P5_L_FOAIE" "breakAfter"
    movej(get_inverse_kin(p[.086035932082, -.461411333971, .148461891445, 1.291226831483, 2.847366049724, -.014272946970], qnear=[1.5120787620544434, -1.655675236378805, 1.688393473625183, -1.61745530763735, -1.5599797407733362, 0.7928479909896851]), a=1.3962634015954636, v=1.0471975511965976)
    $ 456 "Wait: 0.5"
    sleep(0.5)
    $ 457 "MoveL"
    $ 458 "LAS_P5_L_FOAIE" "breakAfter"
    movel(p[.085630803002, -.461977793297, -.018883345701, 1.291225953004, 2.847366487331, -.014272910374], a=1.2, v=0.25)
    $ 459 "Wait: 0.5"
    sleep(0.5)
    $ 460 "'G 80'"
    # 'G 80'
    $ 461 "MoveL"
    $ 462 "DEAS_P5_L" "breakAfter"
    movel(p[.086035888463, -.461411240043, .148461824649, 1.291226985649, 2.847366358337, -.014269561250], a=1.2, v=0.25)
  end
  def Umplu_P4_L():
    $ 463 "Umplu_P4_L" "noBreak"
    $ 464 "MoveJ"
    $ 465 "INTERM_P4" "breakAfter"
    movej(get_inverse_kin(p[-.167567487318, -.286498978533, .168810821008, 1.290941150555, 2.847903107563, -.014389347024], qnear=[0.6869624853134155, -1.9919636885272425, 1.8788256645202637, -1.4593976179706019, -1.5535171667682093, -0.03263694444765264]), a=1.3962634015954636, v=1.0471975511965976)
    $ 466 "Wait: 0.5"
    sleep(0.5)
    $ 467 "MoveJ"
    $ 468 "DEAS_C4_L" "breakAfter"
    movej(get_inverse_kin(p[-.634048678821, .166752753814, .111017315668, 1.076095386128, 2.388610774545, 1.006493672938], qnear=[-0.13465482393373662, -0.5505560080157679, 0.2975288927555084, -0.7133148352252405, -2.1372297445880335, -0.6779091993915003]), a=1.3962634015954636, v=1.0471975511965976)
    $ 469 "Wait: 0.5"
    sleep(0.5)
    $ 470 "MoveL"
    $ 471 "PREL_C4_L" "breakAfter"
    movel(p[-.580966948563, .215040941302, .041371233320, 1.076095361124, 2.388610928008, 1.006493864198], a=1.2, v=0.25)
    $ 472 "Wait: 0.5"
    sleep(0.5)
    $ 473 "'G40'"
    # 'G40'
    $ 474 "MoveL"
    $ 475 "DEAS_C4_LL" "breakAfter"
    movel(p[-.634048678821, .166752753814, .111017315668, 1.076095386128, 2.388610774545, 1.006493672938], a=1.2, v=0.25)
    $ 476 "Wait: 0.5"
    sleep(0.5)
    $ 477 "MoveJ"
    $ 478 "INTER" "breakAfter"
    movej(get_inverse_kin(p[-.167567487318, -.286498978533, .168810821008, 1.290941150555, 2.847903107563, -.014389347024], qnear=[0.6869624853134155, -1.9919636885272425, 1.8788256645202637, -1.4593976179706019, -1.5535171667682093, -0.03263694444765264]), a=1.3962634015954636, v=1.0471975511965976)
    $ 479 "Wait: 0.5"
    sleep(0.5)
    $ 480 "MoveJ"
    $ 481 "DEAS_P4_L_FOAIE" "breakAfter"
    movej(get_inverse_kin(p[.123438262535, -.428229695933, .148259123803, 2.983706482266, .973287546073, -.005232431542], qnear=[1.6059134006500244, -1.7026327292071741, 1.727821707725525, -1.5999348799334925, -1.5731294790851038, 2.546069860458374]), a=1.3962634015954636, v=1.0471975511965976)
    $ 482 "Wait: 0.5"
    sleep(0.5)
    $ 483 "MoveL"
    $ 484 "LAS_P4_L_FOAIE" "breakAfter"
    movel(p[.123033256910, -.428796303747, -.019086199425, 2.983706953586, .973287316837, -.005231605546], a=1.2, v=0.25)
    $ 485 "Wait: 0.5"
    sleep(0.5)
    $ 486 "'G 80'"
    # 'G 80'
    $ 487 "MoveL"
    $ 488 "DEAS_P4_L" "breakAfter"
    movel(p[.123438312068, -.428229638066, .148259065609, 2.983706648639, .973287403808, -.005232379115], a=1.2, v=0.25)
  end
  def UMPLE_P3_L():
    $ 489 "UMPLE_P3_L" "noBreak"
    $ 490 "MoveJ"
    $ 491 "INTERM_P3" "breakAfter"
    movej(get_inverse_kin(p[-.167567487318, -.286498978533, .168810821008, 1.290941150555, 2.847903107563, -.014389347024], qnear=[0.6869624853134155, -1.9919636885272425, 1.8788256645202637, -1.4593976179706019, -1.5535171667682093, -0.03263694444765264]), a=1.3962634015954636, v=1.0471975511965976)
    $ 492 "Wait: 0.5"
    sleep(0.5)
    $ 493 "MoveJ"
    $ 494 "DEAS_C3_L" "breakAfter"
    movej(get_inverse_kin(p[-.634048678821, .166752753814, .111017315668, 1.076095386128, 2.388610774545, 1.006493672938], qnear=[-0.13465482393373662, -0.5505560080157679, 0.2975288927555084, -0.7133148352252405, -2.1372297445880335, -0.6779091993915003]), a=1.3962634015954636, v=1.0471975511965976)
    $ 495 "Wait: 0.5"
    sleep(0.5)
    $ 496 "MoveL"
    $ 497 "PREL_C3_L" "breakAfter"
    movel(p[-.580966948563, .215040941302, .041371233320, 1.076095361124, 2.388610928008, 1.006493864198], a=1.2, v=0.25)
    $ 498 "Wait: 0.5"
    sleep(0.5)
    $ 499 "'G40'"
    # 'G40'
    $ 500 "MoveL"
    $ 501 "DEAS_C3_LL" "breakAfter"
    movel(p[-.634048678821, .166752753814, .111017315668, 1.076095386128, 2.388610774545, 1.006493672938], a=1.2, v=0.25)
    $ 502 "Wait: 0.5"
    sleep(0.5)
    $ 503 "MoveJ"
    $ 504 "INTERMMM" "breakAfter"
    movej(get_inverse_kin(p[-.167567487318, -.286498978533, .168810821008, 1.290941150555, 2.847903107563, -.014389347024], qnear=[0.6869624853134155, -1.9919636885272425, 1.8788256645202637, -1.4593976179706019, -1.5535171667682093, -0.03263694444765264]), a=1.3962634015954636, v=1.0471975511965976)
    $ 505 "Wait: 0.5"
    sleep(0.5)
    $ 506 "MoveJ"
    $ 507 "DEAS_P3_L_FOAIE" "breakAfter"
    movej(get_inverse_kin(p[.156620287324, -.465632395904, .148305405718, 2.983706451876, .973287436954, -.005232257173], qnear=[1.6731274127960205, -1.5915244261371058, 1.6257290840148926, -1.6087849775897425, -1.5733893553363245, 2.613283634185791]), a=1.3962634015954636, v=1.0471975511965976)
    $ 508 "Wait: 0.5"
    sleep(0.5)
    $ 509 "MoveL"
    $ 510 "LAS_P3_L_FOAIE" "breakAfter"
    movel(p[.156215191036, -.466198886150, -.019039951524, 2.983707132669, .973287470355, -.005231765226], a=1.2, v=0.25)
    $ 511 "Wait: 0.5"
    sleep(0.5)
    $ 512 "'G 80'"
    # 'G 80'
    $ 513 "MoveL"
    $ 514 "DEASUPRA_P3_L" "breakAfter"
    movel(p[.156620338377, -.465632333860, .148305347544, 2.983706620081, .973287295311, -.005232216940], a=1.2, v=0.25)
  end
  def Umple_P2_L():
    $ 515 "Umple_P2_L" "noBreak"
    $ 516 "MoveJ"
    $ 517 "interm_P2" "breakAfter"
    movej(get_inverse_kin(p[-.167567487318, -.286498978533, .168810821008, 1.290941150555, 2.847903107563, -.014389347024], qnear=[0.6869624853134155, -1.9919636885272425, 1.8788256645202637, -1.4593976179706019, -1.5535171667682093, -0.03263694444765264]), a=1.3962634015954636, v=1.0471975511965976)
    $ 518 "Wait: 0.5"
    sleep(0.5)
    $ 519 "MoveJ"
    $ 520 "DEAS_cub_C2_L" "breakAfter"
    movej(get_inverse_kin(p[-.634048678821, .166752753814, .111017315668, 1.076095386128, 2.388610774545, 1.006493672938], qnear=[-0.13465482393373662, -0.5505560080157679, 0.2975288927555084, -0.7133148352252405, -2.1372297445880335, -0.6779091993915003]), a=1.3962634015954636, v=1.0471975511965976)
    $ 521 "Wait: 0.5"
    sleep(0.5)
    $ 522 "MoveL"
    $ 523 "prel_c2_L" "breakAfter"
    movel(p[-.580966948563, .215040941302, .041371233320, 1.076095361124, 2.388610928008, 1.006493864198], a=1.2, v=0.25)
    $ 524 "Wait: 0.5"
    sleep(0.5)
    $ 525 "'G40'"
    # 'G40'
    $ 526 "MoveL"
    $ 527 "deas_c2_L" "breakAfter"
    movel(p[-.634048678821, .166752753814, .111017315668, 1.076095386128, 2.388610774545, 1.006493672938], a=1.2, v=0.25)
    $ 528 "Wait: 0.5"
    sleep(0.5)
    $ 529 "MoveJ"
    $ 530 "INTERM" "breakAfter"
    movej(get_inverse_kin(p[-.167567487318, -.286498978533, .168810821008, 1.290941150555, 2.847903107563, -.014389347024], qnear=[0.6869624853134155, -1.9919636885272425, 1.8788256645202637, -1.4593976179706019, -1.5535171667682093, -0.03263694444765264]), a=1.3962634015954636, v=1.0471975511965976)
    $ 531 "Wait: 0.5"
    sleep(0.5)
    $ 532 "MoveJ"
    $ 533 "DEAS_P2_L_FOAIE" "breakAfter"
    movej(get_inverse_kin(p[.189802212420, -.503034964239, .148351669712, 2.983706641880, .973287593777, -.005232243022], qnear=[1.729036569595337, -1.4797232786761683, 1.5095137357711792, -1.6042197386371058, -1.5735967795001429, 2.6691925525665283]), a=1.3962634015954636, v=1.0471975511965976)
    $ 534 "Wait: 0.5"
    sleep(0.5)
    $ 535 "MoveL"
    $ 536 "LAS_P2_L_FOAIE" "breakAfter"
    movel(p[.189397224547, -.503601566376, -.018993557243, 2.983706841452, .973287468046, -.005231518421], a=1.2, v=0.25)
    $ 537 "Wait: 0.5"
    sleep(0.5)
    $ 538 "'G 80'"
    # 'G 80'
    $ 539 "MoveL"
    $ 540 "DEAS_P2_L" "breakAfter"
    movel(p[.189802265547, -.503034898758, .148351611537, 2.983706811229, .973287452528, -.005232213070], a=1.2, v=0.25)
  end
  def Umple_P1_L():
    $ 541 "Umple_P1_L" "noBreak"
    $ 542 "MoveJ"
    $ 543 "Intermediar_cub" "breakAfter"
    movej(get_inverse_kin(p[-.167567487318, -.286498978533, .168810821008, 1.290941150555, 2.847903107563, -.014389347024], qnear=[0.6869624853134155, -1.9919636885272425, 1.8788256645202637, -1.4593976179706019, -1.5535171667682093, -0.03263694444765264]), a=1.3962634015954636, v=1.0471975511965976)
    $ 544 "Wait: 0.5"
    sleep(0.5)
    $ 545 "MoveJ"
    $ 546 "cb_deas_fo_cent" "breakAfter"
    movej(get_inverse_kin(p[.222984199935, -.540437494612, .148398036742, 2.983706804342, .973287476729, -.005232058460], qnear=[1.7761387825012207, -1.3659704367267054, 1.3774471282958984, -1.5857699553119105, -1.5737646261798304, 2.716294765472412]), a=1.3962634015954636, v=1.0471975511965976)
    $ 547 "Wait: 0.5"
    sleep(0.5)
    $ 548 "MoveL"
    $ 549 "las_1_cub_foaie" "breakAfter"
    movel(p[.222579162379, -.541004135262, -.018947151668, 2.983706805502, .973287480323, -.005231718426], a=1.2, v=0.25)
    $ 550 "Wait: 0.5"
    sleep(0.5)
    $ 551 "'G 80'"
    # 'G 80'
    $ 552 "MoveL"
    $ 553 "Deasupra_foaiee" "breakAfter"
    movel(p[.222984255685, -.540437426381, .148397978555, 2.983706974383, .973287335722, -.005232037241], a=1.2, v=0.25)
  end
  def Deasupra_cuburi():
    $ 554 "Deasupra_cuburi" "noBreak"
    $ 555 "MoveL"
    $ 556 "DeasupraMarker2" "breakAfter"
    movel(p[-.167556988585, -.286490343035, .168794710650, 1.290935638895, 2.847889630710, -.014342479944], a=1.2, v=0.25)
    $ 557 "MoveJ"
    $ 558 "poz_intermcub" "breakAfter"
    movej(get_inverse_kin(p[-.634048678821, .166752753814, .111017315668, 1.076095386128, 2.388610774545, 1.006493672938], qnear=[-0.13465482393373662, -0.5505560080157679, 0.2975288927555084, -0.7133148352252405, -2.1372297445880335, -0.6779091993915003]), a=1.3962634015954636, v=1.0471975511965976)
    $ 559 "MoveL"
    $ 560 "prindere_cub" "breakAfter"
    movel(p[-.580966948563, .215040941302, .041371233320, 1.076095361124, 2.388610928008, 1.006493864198], a=1.2, v=0.25)
    $ 561 "Wait: 0.5"
    sleep(0.5)
    $ 562 "'G40'"
    # 'G40'
    $ 563 "MoveL"
    $ 564 "poz_intermcub" "breakAfter"
    movel(p[-.634048678821, .166752753814, .111017315668, 1.076095386128, 2.388610774545, 1.006493672938], a=1.2, v=0.25)
    $ 565 "Wait: 0.5"
    sleep(0.5)
  end
  def Lasa_Marker_Poz_cub():
    $ 566 "Lasa_Marker_Poz_cub" "noBreak"
    $ 567 "MoveL"
    $ 568 "DeasupraFoaie" "breakAfter"
    movel(p[.256474810278, -.543503263666, .147758605300, 1.296043006987, 2.848526747641, .014472740185], a=1.2, v=0.25)
    $ 569 "MoveJ"
    $ 570 "DeasupraMarker" "breakAfter"
    movej(get_inverse_kin(p[-.167556988585, -.286490343035, .168794710650, 1.290935638895, 2.847889630710, -.014342479944], qnear=[0.6869624257087708, -1.991971794758932, 1.8788633346557617, -1.4593938032733362, -1.5535171667682093, -0.03263694444765264]), a=1.3962634015954636, v=1.0471975511965976)
    $ 571 "MoveL"
    $ 572 "LasaMarker" "breakAfter"
    movel(p[-.167798968899, -.286828969517, .068795580420, 1.290935342563, 2.847889621865, -.014342483373], a=1.2, v=0.25)
    $ 573 "Wait: 0.5"
    sleep(0.5)
    $ 574 "'G 40'"
    # 'G 40'
    $ 575 "Wait: 0.5"
    sleep(0.5)
    $ 576 "MoveL"
    $ 577 "DeasupraMarker2" "breakAfter"
    movel(p[-.167556988585, -.286490343035, .168794710650, 1.290935638895, 2.847889630710, -.014342479944], a=1.2, v=0.25)
    $ 578 "Wait: 0.5"
    sleep(0.5)
    $ 579 "'G80'"
    # 'G80'
  end
  def Desen_L():
    $ 580 "Desen_L" "noBreak"
    $ 581 "MoveL"
    $ 582 "exterior_L" "breakAfter"
    movel(p[.125171699055, -.392752669928, .047564988851, 1.296043247772, 2.848527468985, .014471667445], a=1.2, v=0.25)
    $ 583 "MoveL"
    $ 584 "Exterior_L2" "breakAfter"
    movel(p[.012964415184, -.492297288535, .048173660313, 1.296043209345, 2.848527577839, .014472062410], a=1.2, v=0.25)
    $ 585 "MoveL"
    $ 586 "Exterior_L3" "breakAfter"
    movel(p[.046146443999, -.529699809471, .048219926550, 1.296043240397, 2.848527550464, .014472614211], a=1.2, v=0.25)
    $ 587 "MoveL"
    $ 588 "Interior_L" "breakAfter"
    movel(p[.120039742713, -.464145300243, .047818946711, 1.296043304535, 2.848527608211, .014473209978], a=1.2, v=0.25)
    $ 589 "MoveL"
    $ 590 "Interior_L2" "breakAfter"
    movel(p[.219585684133, -.576353078437, .047957978891, 1.296043281349, 2.848527543905, .014473409645], a=1.2, v=0.25)
    $ 591 "MoveL"
    $ 592 "Interior_L3" "breakAfter"
    movel(p[.256232678162, -.543841851762, .047759338732, 1.296043088135, 2.848527130158, .014473054523], a=1.2, v=0.25)
  end
  while (True):
    $ 1 "Robot Program"
    $ 2 "MoveL"
    $ 3 "Intermediar_cub" "breakAfter"
    movel(p[-.167567487318, -.286498978533, .168810821008, 1.290941150555, 2.847903107563, -.014389347024], a=1.2, v=0.25)
    $ 4 "preluare_marker" "breakAfter"
    movel(p[-.167809654265, -.286837740331, .068811761063, 1.290941692887, 2.847902933041, -.014390023281], a=1.2, v=0.25)
    $ 5 "Wait: 0.5"
    sleep(0.5)
    $ 6 "'G 10'"
    # 'G 10'
    $ 7 "Wait: 0.5"
    sleep(0.5)
    $ 8 "MoveL"
    $ 9 "ridicare_marker" "breakAfter"
    movel(p[-.167567662759, -.286499098442, .168810924250, 1.290942013576, 2.847902999547, -.014390179140], a=1.2, v=0.25)
    $ 10 "MoveJ"
    $ 11 "deasupra_colt_f" "breakAfter"
    movej(get_inverse_kin(p[.258141789851, -.542024496562, .147749670065, 1.296043017352, 2.848526902154, .014471210395], qnear=[1.8233630657196045, -1.3276937643634241, 1.330954670906067, -1.5744360128985804, -1.5556119124041956, 1.1065565347671509]), a=1.3962634015954636, v=1.0471975511965976)
    $ 12 "MoveL"
    $ 13 "marker_pe_colt" "breakAfter"
    movel(p[.257899646872, -.542363131498, .047750427825, 1.296043067917, 2.848527220905, .014471310607], a=1.2, v=0.25)
    $ 14 "If digital_in[1] == True"
    if (digital_in[1] == True):
      $ 15 "Call Desen_L"
      Desen_L()
      $ 16 "Call Lasa_Marker_Poz_cub"
      Lasa_Marker_Poz_cub()
      $ 17 "Call Deasupra_cuburi"
      Deasupra_cuburi()
      $ 18 "Call Umple_P1_L"
      Umple_P1_L()
      $ 19 "Call Umple_P2_L"
      Umple_P2_L()
      $ 20 "Call UMPLE_P3_L"
      UMPLE_P3_L()
      $ 21 "Call Umplu_P4_L"
      Umplu_P4_L()
      $ 22 "Call Umplu_P5_L"
      Umplu_P5_L()
      $ 23 "Call Umplu_P6_L"
      Umplu_P6_L()
    end
    $ 24 "If digital_in[2] ==  True "
    if (get_standard_digital_in(2) ==   True  ):
      $ 25 "Call Desen_i"
      Desen_i()
      $ 26 "Call Lasa_Marker_Poz_cub"
      Lasa_Marker_Poz_cub()
      $ 27 "Call Deasupra_cuburi"
      Deasupra_cuburi()
      $ 28 "Call Umple_P1_L"
      Umple_P1_L()
      $ 29 "Call Umplu_p2_i"
      Umplu_p2_i()
      $ 30 "Call Umplu_p3_i"
      Umplu_p3_i()
    end
    $ 31 "If digital_in[3] ==  True "
    if (get_standard_digital_in(3) ==   True  ):
      $ 32 "Call Desen_H"
      Desen_H()
      $ 33 "Call Lasa_Marker_Poz_cub"
      Lasa_Marker_Poz_cub()
      $ 34 "Call Deasupra_cuburi"
      Deasupra_cuburi()
      $ 35 "Call Umple_P1_L"
      Umple_P1_L()
      $ 36 "Call Umple_P2_L"
      Umple_P2_L()
      $ 37 "Call UMPLE_P3_L"
      UMPLE_P3_L()
      $ 38 "Call Umple_P4_H"
      Umple_P4_H()
      $ 39 "Call Umple_P5_H"
      Umple_P5_H()
      $ 40 "Call Umple_P6_H"
      Umple_P6_H()
      $ 41 "Call Umple_P7_H"
      Umple_P7_H()
    end
    $ 42 "If digital_in[5] ==  True "
    if (get_standard_digital_in(5) ==   True  ):
      $ 43 "Call Desen_T"
      Desen_T()
      $ 44 "Call Lasa_Marker_Poz_cub"
      Lasa_Marker_Poz_cub()
      $ 45 "Call Deasupra_cuburi"
      Deasupra_cuburi()
      $ 46 "Call Umple_P1_L"
      Umple_P1_L()
      $ 47 "Call Umple_P2_T"
      Umple_P2_T()
      $ 48 "Call Umple_p3_T"
      Umple_p3_T()
      $ 49 "Call Umplu_p4_t"
      Umplu_p4_t()
      $ 50 "Call Umplu_p5_T"
      Umplu_p5_T()
      $ 51 "Call Umple_P6_T"
      Umple_P6_T()
    end
  end
end
